DATA_BLOCK "DB_MVD_Type"
TITLE =%version: 0.13 % CN: 20
//History:
//This version  %created_by: nlhdl %
//              %date_created: Friday, December 08, 2017 2:58:35 PM %
//              %release: VI_RAW/RA_Dev %
//
//Modification History:                                   By:    Date:     Rev:
//----------------------------------------------------  -------  --------  -----
//ra#26909: general state Redundancy to warning         nlHdL    08-12-17   0.13
//ra#24205:Align Bits for HMI Zone                      inajos   09-11-17   0.12
//bhs#18875: MVD Add switch fieldbus slave              nlHdL    22-05-17   0.11
//ra#18174: DI NON_RETAIN PLC Memory                    nlHdL    14-12-16   0.10
//ra#15770: Update because of change in statussen       nlJClo   21-07-16   0.09
//ra#15770: Update the MVD according MCFV decomposition nlHdL    18-07-16   0.08
//ra#15770: Update the MVD according MCFV decomposition nlHdL    18-07-16   0.08
//7324: ECS-P General from the RD to RA for platform    nlHdL    06-07-15   0.08
//21030: Markcode change SVZ MVZ to SVD MVD             nlHdL    24-09-14   0.08
//16446: Rework to make consequent with SVZ             nlple    06-12-13   0.07
//16446: Overal/general status 1/6/11 changed           nlple    06-12-13   0.06
//15797: Keyword release added                          nlwwij   26-09-13   0.05
//CR10485 Removed comment from type DB                  nlHHop   25-06-12   0.04
//CR8713 Changing after test on site                    nlple    10-01-12   0.03
//CR7783 modified general & overal status 11,13 and 14  nlHHop   22-09-11   0.02
//Initial revision                                      nlLvdG   22-10-10   0.01
//
FAMILY : RAW
VERSION : 0.0
NON_RETAIN


 STRUCT
   Type_Component : BYTE ;	//Type of the component (1 = Section, 0 = Other)
   Record_Length : BYTE ;	//Number of the Detailed Status in the UDT
   Status : ARRAY  [1 .. 16 ] OF "UDT_Comp_Status";
  END_STRUCT ;
BEGIN
   Type_Component := B#16#0;
   Record_Length := B#16#16;
   Status[1].HMI_Text_Number := -1;
   Status[1].Overall_Status_Relation := B#16#1;
   Status[1].General_Status_Relation := B#16#4;
   Status[2].HMI_Text_Number := -1;
   Status[2].Overall_Status_Relation := B#16#1;
   Status[2].General_Status_Relation := B#16#4;
   Status[3].HMI_Text_Number := -1;
   Status[3].Overall_Status_Relation := B#16#2;
   Status[3].General_Status_Relation := B#16#2;
   Status[4].HMI_Text_Number := 47;
   Status[4].Overall_Status_Relation := B#16#2;
   Status[4].General_Status_Relation := B#16#2;
   Status[5].HMI_Text_Number := 60;
   Status[5].Overall_Status_Relation := B#16#4;
   Status[5].General_Status_Relation := B#16#3;
   Status[6].HMI_Text_Number := 61;
   Status[6].Overall_Status_Relation := B#16#4;
   Status[6].General_Status_Relation := B#16#3;
   Status[7].HMI_Text_Number := 31;
   Status[7].Overall_Status_Relation := B#16#4;
   Status[7].General_Status_Relation := B#16#3;
   Status[8].HMI_Text_Number := -1;
   Status[8].Overall_Status_Relation := B#16#0;
   Status[8].General_Status_Relation := B#16#0;
   Status[9].HMI_Text_Number := -1;
   Status[9].Overall_Status_Relation := B#16#0;
   Status[9].General_Status_Relation := B#16#0;
   Status[10].HMI_Text_Number := -1;
   Status[10].Overall_Status_Relation := B#16#0;
   Status[10].General_Status_Relation := B#16#0;
   Status[11].HMI_Text_Number := -1;
   Status[11].Overall_Status_Relation := B#16#0;
   Status[11].General_Status_Relation := B#16#0;
   Status[12].HMI_Text_Number := 280;
   Status[12].Overall_Status_Relation := B#16#4;
   Status[12].General_Status_Relation := B#16#3;
   Status[13].HMI_Text_Number := 281;
   Status[13].Overall_Status_Relation := B#16#4;
   Status[13].General_Status_Relation := B#16#3;
   Status[14].HMI_Text_Number := -1;
   Status[14].Overall_Status_Relation := B#16#0;
   Status[14].General_Status_Relation := B#16#0;
   Status[15].HMI_Text_Number := -1;
   Status[15].Overall_Status_Relation := B#16#0;
   Status[15].General_Status_Relation := B#16#0;
   Status[16].HMI_Text_Number := -1;
   Status[16].Overall_Status_Relation := B#16#0;
   Status[16].General_Status_Relation := B#16#0;
END_DATA_BLOCK

